// TwinCAT 3 PLC project OEF_9
// ProgramVersion: 3.1.4024.0
// libraries:
//   Tc2_Standard, * (Beckhoff Automation GmbH)
//   Tc2_System, * (Beckhoff Automation GmbH)
//   Tc3_Module, * (Beckhoff Automation GmbH)
// project tree:
//   / GlobalTextList.TcGTLO, PlcTask.TcTTO, Visualization Manager.TcVMO (not stored)
//   POUs/ MAIN.TcPOU
//   VISUs/ Visualization.TcVIS
// (motion and I/O tree: see PLC project oef_1)
// real-time tasks:
//   TASK PlcTask: cycle T#10ms, priority 20, ADS port 350
//   TASK PlcTask1: cycle T#10ms, priority 21, ADS port 351
//   TASK PlcTask2: cycle T#10ms, priority 22, ADS port 352
//   TASK PlcTask3: cycle T#10ms, priority 23, ADS port 353
//   TASK PlcTask4: cycle T#10ms, priority 24, ADS port 354
//   TASK PlcTask5: cycle T#10ms, priority 25, ADS port 355
//   TASK PlcTask6: cycle T#10ms, priority 26, ADS port 356
// variable links:

CONFIGURATION OEF_9
    RESOURCE PLC ON TwinCAT3
        TASK PlcTask(INTERVAL := T#10ms, PRIORITY := 26);
        PROGRAM MAIN WITH PlcTask : MAIN;
    END_RESOURCE
END_CONFIGURATION

// ---- POUs/MAIN.TcPOU
PROGRAM MAIN
VAR
	TotalOutput AT %Q*: INT;
	Vat1 AT %I*: INT := 0;
	Vat2 AT %I*: INT := 0;
	Vat3 AT %I*: INT := 0;
END_VAR

TotalOutput := (Vat1 + Vat2 + Vat3);

END_PROGRAM

// ---- VISUs/Visualization.TcVIS
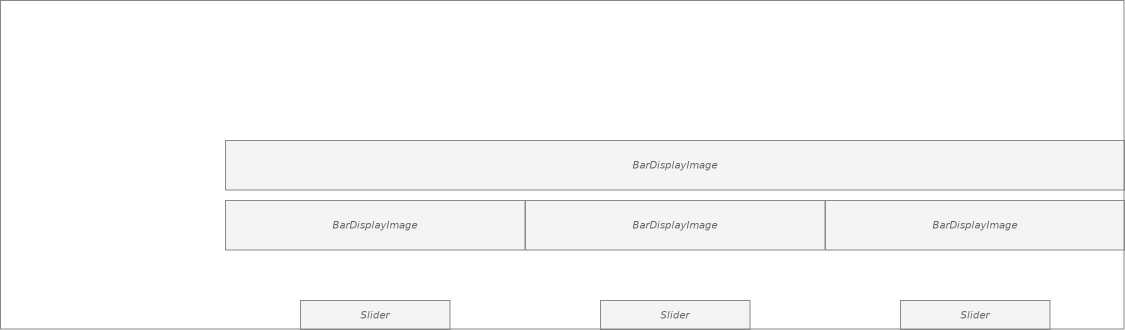
VISUALIZATION Visualization  // 1125x330
    Slider (600,300 150x30), variable: MAIN.Vat2, scale 0..3000
    Slider (900,300 150x30), variable: MAIN.Vat3, scale 0..5000
    Slider (300,300 150x30), variable: MAIN.Vat1, scale 0..2000
    BarDisplayImage (225,200 300x50), value: MAIN.Vat1, style: BarDisplayImage-Gray, scale format: %.1f, scale 0..2000
    BarDisplayImage (525,200 300x50), value: MAIN.Vat2, style: BarDisplayImage-Gray, scale format: %.1f, scale 0..3000
    BarDisplayImage (825,200 300x50), value: MAIN.Vat3, style: BarDisplayImage-Gray, scale format: %.1f, scale 0..5000
    BarDisplayImage (225,140 900x50), value: MAIN.TotalOutput, style: BarDisplayImage-Gray, scale format: %.1f, scale 0..10000
END_VISUALIZATION
